// TIA Portal V20 export
VAR_GLOBAL   // PLC tag table "Default tag table"
   Start AT %I0.0 : Bool;
   Stop AT %I0.1 : Bool;
   ProgramOn AT %I0.2 : Bool;
END_VAR
